FUNCTION_BLOCK TIMER_ALARM
VAR_INPUT
	BOOL_SIGNAL_IN: BOOL;
	BOOL_ALMRST_PB: BOOL;
	BOOL_BZRST_PB: BOOL;
	INT_PV: INT;

END_VAR

VAR_OUTPUT
	ALM_MSG_BOOL: BOOL;
	BZ_OUT_BOOL: BOOL;
	EV_INT: INT;
END_VAR

VAR
	T1: TON;
	M0: BOOL;
	M1: BOOL;
	D200: TIME;
	D202: INT;
END_VAR

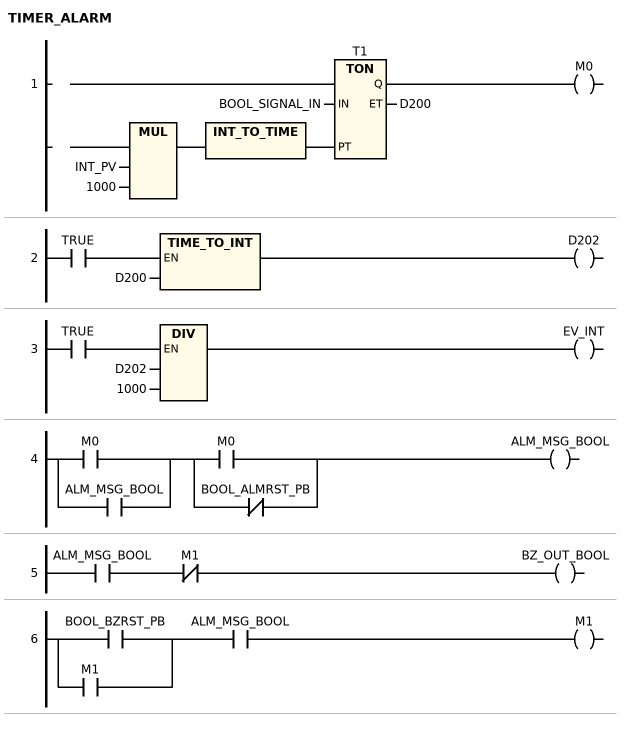
// NETWORK 1
T1(IN := BOOL_SIGNAL_IN, PT := INT_TO_TIME(INT_PV * 1000), ET => D200); // TON
M0 := T1.Q;

// NETWORK 2
D202 := TIME_TO_INT(D200);

// NETWORK 3
EV_INT := D202 / 1000;

// NETWORK 4
ALM_MSG_BOOL := (M0 OR ALM_MSG_BOOL) AND (M0 OR NOT BOOL_ALMRST_PB);

// NETWORK 5
BZ_OUT_BOOL := ALM_MSG_BOOL AND NOT M1;

// NETWORK 6
M1 := (BOOL_BZRST_PB OR M1) AND ALM_MSG_BOOL;

END_FUNCTION_BLOCK

(* stored: Version 1.1.0.1, ProductVersion 3.1.4024.12
   POU TIMER_ALARM: Id {8ad684c6-774e-43c2-a1dd-17ff0cf67b1d}, SpecialFunc None *)
